FUNCTION_BLOCK FB_ProBoxElementMotor EXTENDS FB_ProBoxElementBase
(**************************************************************************************
 * 	Application		:	BoxControl Framework
 *	Revision		:	$Revision: $
 *	Revision date	:	$Date: $
 *	Last changed by	:	$Author:  $
 *	URL				:	$URL: $
 *
 *	Purpose			:	ProBox element with one drive.
 *
 * ------------------------------------------------------------------------------------
 *	Copyright Swisslog [IP AG], Switzerland. All rights reserved.
 * 
 * ------------------------------------------------------------------------------------
 *	
 * 	Revision History: 
 *
 * 	VERSION			DATE			INITIALS			DESCRIPTION
  *
 **************************************************************************************)
VAR_INPUT
	Config					: ST_CFG_ProBoxElementMotor; // Configuration	
	HW_Inputs				: ST_HW_InputsProBoxElementMotor; // HW-Inputs	
END_VAR

VAR_OUTPUT
	HW_Outputs				: ST_HW_OutputsProBoxElementMotor; // HW-Outputs
END_VAR


VAR PERSISTENT
	Settings				: ST_CFG_ProBoxElementMotor; // Settings - activated configuration 
END_VAR


(**************************************************************************************************************
   Input mapping
***************************************************************************************************************)
A_InputMapping();


(**************************************************************************************************************
   Initialization
***************************************************************************************************************)
A_Init();


(**************************************************************************************************************
   State control
***************************************************************************************************************)
A_StateControl();


(**************************************************************************************************************
   Error handler
***************************************************************************************************************)
M_MonitorElementErrors();


(**************************************************************************************************************
   Manual control
***************************************************************************************************************)
A_ManualControl();


(**************************************************************************************************************
   Handle element functions
***************************************************************************************************************)
A_HandleFunctions();


(**********************************************************************************************************
   Drive control
***********************************************************************************************************)

A_DriveControl();



(**************************************************************************************************************
   Interface handler out
***************************************************************************************************************)
M_ITC_ProcessOut();


(**************************************************************************************************************
   Output mapping
***************************************************************************************************************)
A_OutputMapping();

ACTION A_Init:
(**************************************************************************************
 * 	NAME		A_Init
 * 	FUNCTION	Initialize element
 **************************************************************************************)

 
 
 IF NOT ElementData.Init AND NOT ElementData.InitRunning THEN
	 // Load function specific configuration to settings
	Settings := Config;
	SUPER^.BaseSettings.BrakeTime := Settings.BrakeTime;	
	SUPER^.BaseSettings.ElementSpeed := Settings.ElementSpeed;
 END_IF
 
SUPER^.A_Init();
END_ACTION

ACTION A_InputMapping:
(**************************************************************************************
 * 	NAME		A_InputMapping
 * 	FUNCTION	Input mapping
 **************************************************************************************)
 
 
(**************************************************************************************
   Map HW Inputs
***************************************************************************************)
Inputs.MotorUnitOK := HW_inputs.MotorUnitOK;

SUPER^.A_InputMapping();
END_ACTION

ACTION A_OutputMapping:
(**************************************************************************************
 * 	NAME		A_OutputMapping
 * 	FUNCTION	Handles element specific outpus
 **************************************************************************************)

(**************************************************************************************
   Map HW Outputs
***************************************************************************************)
HW_Outputs.Drive_Run_12		:= fbProBoxMotorControl_12.Forward;
HW_Outputs.Drive_Run_21		:= fbProBoxMotorControl_12.Reverse;
HW_Outputs.Drive_Creep_12	:= fbProBoxMotorControl_12.CreepSpeed;
HW_Outputs.Drive_Low_12		:= fbProBoxMotorControl_12.LowSpeed;
HW_Outputs.MotorBrake_12	:= fbProBoxMotorControl_12.BrakeRelease;


Super^.A_OutputMapping();
END_ACTION

END_FUNCTION_BLOCK

(* stored: Version 1.1.0.1, ProductVersion 3.1.4024.9
   POU FB_ProBoxElementMotor: Id {0b822cdd-9b0a-4f15-b748-e8b3e1b8258b}, SpecialFunc None
   Action A_Init: Id {e3e50279-f341-4b4a-a77c-accead4d286a}
   Action A_InputMapping: Id {217bdc6a-cf49-41be-a409-75a25ac4cfa8}
   Action A_OutputMapping: Id {fc78955c-d744-4913-a6c9-6c39824b616b} *)
